Staubli VAL3: onBackEvent.pgx

program onBackEvent()
  local string l_sItem
  local num i
begin
  //
  // rename
  //
  if nFrame>0
    l_sItem=saveData:fFrameItem[nFrame].sName
    if l_sItem!=""
      i=find(sEvent,l_sItem)
    else
      i=len(toString("",nFrame))+3
    endIf
    if i!=-1
      // clean the line
      call use:listcursor(use:nView,false)
      // read the name
      call use:read(40-use:nBottomX+i-1,nView+1,l_sItem,10,false)
      saveData:fFrameItem[nFrame].sName=l_sItem
      call buildList()
      use:bUseRefresh=true
    endIf
  endIf
end
